% RSLogix 500 project STRINGS PROCESING.RSS, saved by version 8.30.00.16 %
PROJECT "ASCAES"    % processor: Bul.1763 MicroLogix 1100 Series B %

PROGRAM FILES
  LAD 2   14 rungs

DATA FILES
  O0 OUTPUT  4 elements
  I1 INPUT  6 elements
  S2 STATUS  66 elements
  B3 BINARY  1 elements
  T4 TIMER  1 elements
  C5 COUNTER  1 elements
  R6 CONTROL  1 elements
  N7 INTEGER  5 elements
  F8 FLOAT  1 elements
  ST9 STRING  12 elements

LADDER 2
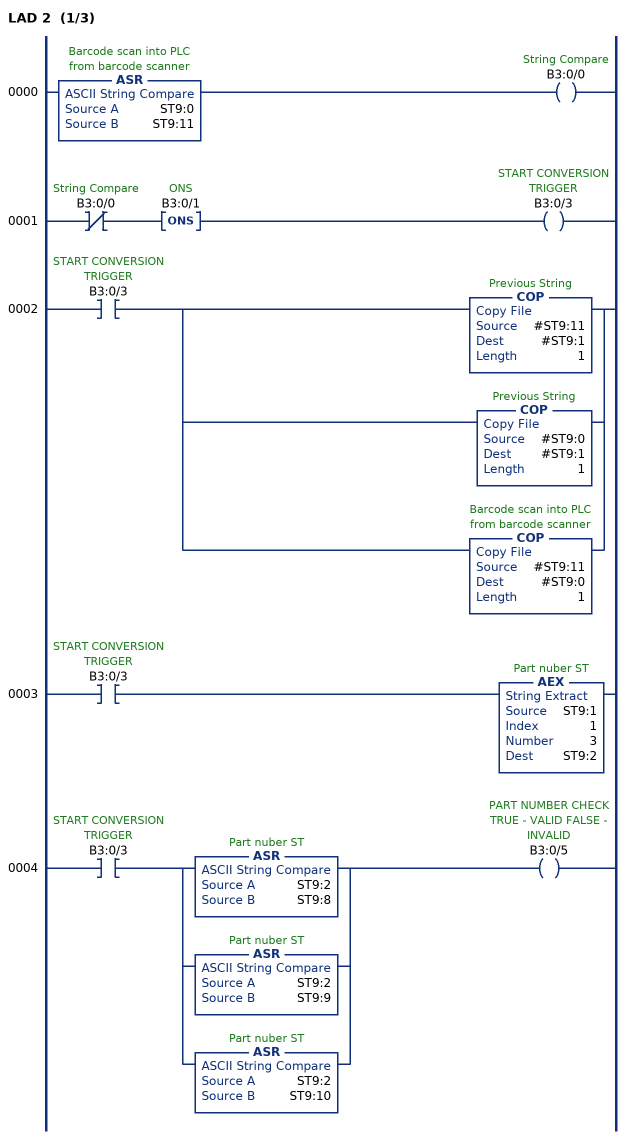
% Rung: 0 %
SOR ASR ST9:0 ST9:11 OTE B3:0/0 EOR
%   ST9:0  "Barcode scan into PLC from barcode scanner" %
%   ST9:11  EMPTY_STR  "EMPTY STRING" %
%   B3:0/0  "String Compare" %
% Rung: 1 %
SOR XIO B3:0/0 ONS B3:0/1 OTE B3:0/3 EOR
%   B3:0/0  "String Compare" %
%   B3:0/1  "ONS" %
%   B3:0/3  "START CONVERSION TRIGGER" %
% Rung: 2 %
SOR XIC B3:0/3 BST COP #ST9:11 #ST9:1 1 NXB COP #ST9:0 #ST9:1 1 NXB COP #ST9:11 #ST9:0 1 BND EOR
%   B3:0/3  "START CONVERSION TRIGGER" %
%   ST9:11  EMPTY_STR  "EMPTY STRING" %
%   ST9:1  "Previous String" %
%   ST9:0  "Barcode scan into PLC from barcode scanner" %
% Rung: 3 %
SOR XIC B3:0/3 AEX ST9:1 1 3 ST9:2 EOR
%   B3:0/3  "START CONVERSION TRIGGER" %
%   ST9:1  "Previous String" %
%   ST9:2  ST  "Part nuber" %
% Rung: 4 %
SOR XIC B3:0/3 BST ASR ST9:2 ST9:8 NXB ASR ST9:2 ST9:9 NXB ASR ST9:2 ST9:10 BND OTE B3:0/5 EOR
%   B3:0/3  "START CONVERSION TRIGGER" %
%   ST9:2  ST  "Part nuber" %
%   ST9:8  "PART NUMBER 123" %
%   ST9:9  "PART NUMBER 456" %
%   ST9:10  "PART NUMBER 789" %
%   B3:0/5  "PART NUMBER CHECK TRUE - VALID FALSE - INVALID" %

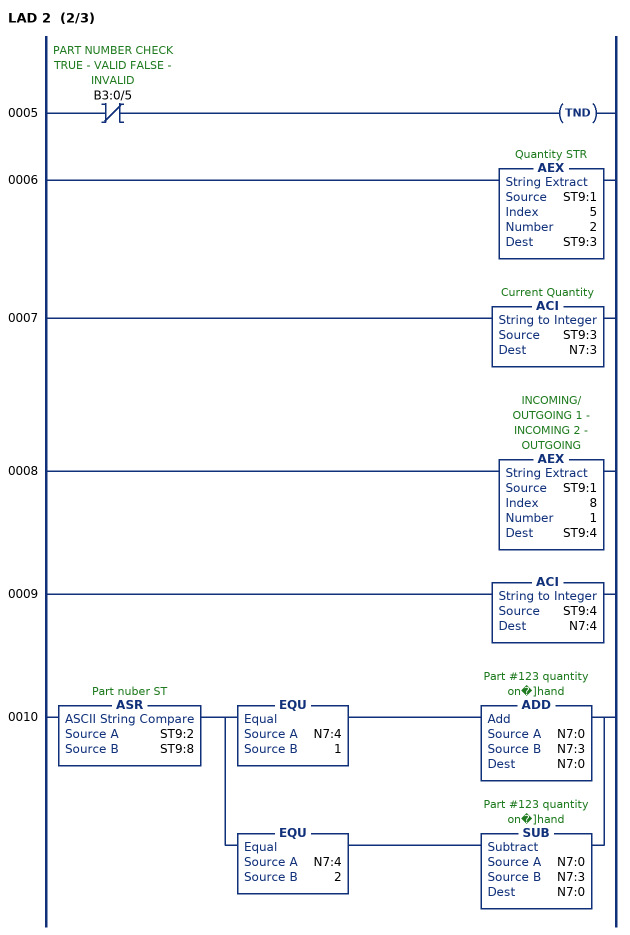
% Rung: 5 %
SOR XIO B3:0/5 TND EOR
%   B3:0/5  "PART NUMBER CHECK TRUE - VALID FALSE - INVALID" %
% Rung: 6 %
SOR AEX ST9:1 5 2 ST9:3 EOR
%   ST9:1  "Previous String" %
%   ST9:3  "Quantity STR" %
% Rung: 7 %
SOR ACI ST9:3 N7:3 EOR
%   ST9:3  "Quantity STR" %
%   N7:3  "Current Quantity" %
% Rung: 8 %
SOR AEX ST9:1 8 1 ST9:4 EOR
%   ST9:1  "Previous String" %
%   ST9:4  "INCOMING/OUTGOING 1 - INCOMING 2 - OUTGOING" %
% Rung: 9 %
SOR ACI ST9:4 N7:4 EOR
%   ST9:4  "INCOMING/OUTGOING 1 - INCOMING 2 - OUTGOING" %
% Rung: 10 %
SOR ASR ST9:2 ST9:8 BST EQU N7:4 1 ADD N7:0 N7:3 N7:0 NXB EQU N7:4 2 SUB N7:0 N7:3 N7:0 BND EOR
%   ST9:2  ST  "Part nuber" %
%   ST9:8  "PART NUMBER 123" %
%   N7:0  "Part #123 quantity on�]hand" %
%   N7:3  "Current Quantity" %

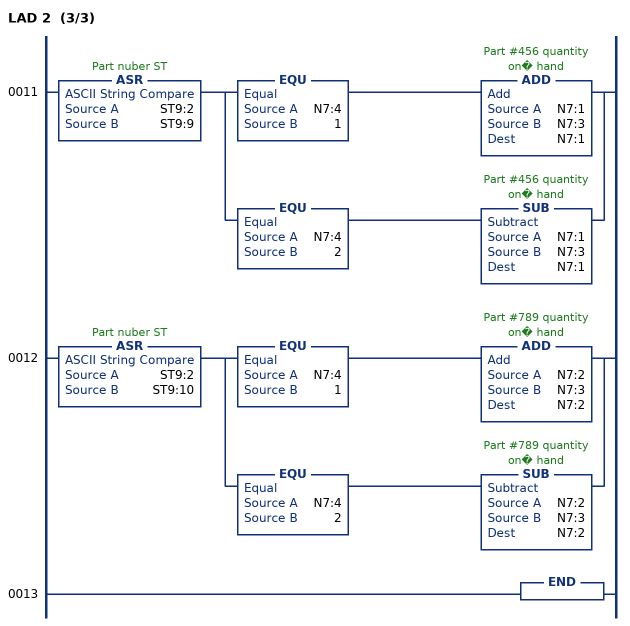
% Rung: 11 %
SOR ASR ST9:2 ST9:9 BST EQU N7:4 1 ADD N7:1 N7:3 N7:1 NXB EQU N7:4 2 SUB N7:1 N7:3 N7:1 BND EOR
%   ST9:2  ST  "Part nuber" %
%   ST9:9  "PART NUMBER 456" %
%   N7:1  "Part #456 quantity on� hand" %
%   N7:3  "Current Quantity" %
% Rung: 12 %
SOR ASR ST9:2 ST9:10 BST EQU N7:4 1 ADD N7:2 N7:3 N7:2 NXB EQU N7:4 2 SUB N7:2 N7:3 N7:2 BND EOR
%   ST9:2  ST  "Part nuber" %
%   ST9:10  "PART NUMBER 789" %
%   N7:2  "Part #789 quantity on� hand" %
%   N7:3  "Current Quantity" %
% Rung: 13 %
SOR END EOR

OTHER DOCUMENTED ADDRESSES
  B3:0/4  "ONS"

DATA TABLE (non-zero values as saved)
DATA B3
% B3:0 % 0X0012
DATA ST9
% ST9:0 % "123-10:1"
% ST9:1 % "789-29-2"
% ST9:2 % "789"
% ST9:3 % "29"
% ST9:4 % "2"
% ST9:8 % "123"
% ST9:9 % "456"
% ST9:10 % "789"
